// TIA Portal V19 export
TYPE "LEXCHANGETRAY_typeRoller_deliver_interface"
// stored: Access Published
   STRUCT
      init : Bool;
      logistics : "LEXCHANGETRAY_typeRoller_toLogisticsDeliver";
      workStationRoller { S7_SetPoint := 'True'} : "LEXCHANGETRAY_typeRoller_toWorkstationDeliver";
   END_STRUCT;
END_TYPE
